{attribute 'qualified_only'}
{attribute 'strict'}
TYPE E_MergeMode :
(
	BlockedWait := 0,
	ChaseTailStatic := 1, //also 'window'
	MergeInAhead := 2 // KeepGoing or from Standstill
);
END_TYPE

(* stored: Version 1.1.0.1
   DUT E_MergeMode: Id {57d55088-9666-061f-0842-13c5b7a7141d} *)
